/// determines whether the actual speed (ABS value) is within the target-speed window
FUNCTION F_SpeedWindowReached : BOOL
VAR_INPUT
	/// factor for tolerance (default: 0.1)
	fToleranceFactor: REAL;
	/// actual speed
	fActualSpeed: LREAL;
	/// target speed
	fTargetSpeed: LREAL;
	/// Override for axis and spindle
	fOverride: LREAL;
END_VAR
VAR CONSTANT
	fDefaultfToleranceFactor: REAL := 0.1;
END_VAR
VAR
	fTol: LREAL;
	fMin: LREAL;
	fMax: LREAL;
	fAct: LREAL;
	fTar: LREAL;
END_VAR

// validate tolerance factor
IF fToleranceFactor <= 0 THEN
	fToleranceFactor:=fDefaultfToleranceFactor;
END_IF

// calc tolerance window and ABS values
fTar:=fTargetSpeed*(fOverride/100);
fTol:=ABS(fTar) * fToleranceFactor;
fMin:=ABS(fTar) - fTol;
fMax:=ABS(fTar) + fTol;
fAct:=ABS(fActualSpeed);

F_SpeedWindowReached := fAct >= fMin AND fAct <= fMax;

END_FUNCTION

(* stored: Version 1.1.0.1, ProductVersion 3.1.4020.12
   POU F_SpeedWindowReached: Id {0d48aba9-7f39-413b-a20f-a6f46ffe621b}, SpecialFunc None *)
